TYPE TupleStruct_5:
    STRUCT
        field0: LREAL;
        field1: LREAL;
        field2: LREAL;
        field3: LREAL;
        field4: LREAL;
        field5: LREAL;
        field6: LREAL;
        field7: LREAL;
        field8: LREAL;
        field9: LREAL;
        field10: LREAL;
        field11: LREAL;
        field12: LREAL;
        field13: LREAL;
        field14: LREAL;
        field15: LREAL;
        field16: LREAL;
        field17: LREAL;
        field18: LREAL;
        field19: LREAL;
        field20: LREAL;
        field21: LREAL;
        field22: LREAL;
        field23: LREAL;
        field24: LREAL;
        field25: LREAL;
        field26: LREAL;
        field27: LREAL;
        field28: LREAL;
        field29: LREAL;
        field30: LREAL;
        field31: LREAL;
        field32: LREAL;
        field33: LREAL;
        field34: LREAL;
        field35: LREAL;
        field36: LREAL;
        field37: LREAL;
        field38: LREAL;
        field39: LREAL;
        field40: LREAL;
        field41: LREAL;
        field42: LREAL;
        field43: LREAL;
        field44: LREAL;
        field45: LREAL;
        field46: LREAL;
        field47: LREAL;
        field48: LREAL;
        field49: LREAL;
        field50: LREAL;
        field51: LREAL;
        field52: LREAL;
        field53: LREAL;
        field54: LREAL;
        field55: LREAL;
        field56: LREAL;
        field57: LREAL;
        field58: LREAL;
    END_STRUCT
END_TYPE

(* stored: ProductVersion 3.1.0.18, Version 1.1.0.1 *)
